// TIA Portal V19 export
TYPE "typeVfdGeneral"
// stored: Access Published
   STRUCT
      acc : Real;   // 手动速度上限
      dec : Real;   // 手动速度设定值，画面做限制根据上限值如果超了不允许输入
      fastdec : Real;
      refSpeed : Real;
      simActive : Bool;   // Manual mode parameters for axis control interface
   END_STRUCT;
END_TYPE
